TYPE
    ST_PickPlaceDetail : STRUCT
        MemberType : STRING;
        XPos       : REAL;
        YPos       : REAL;
        ZPos       : REAL;
        ZRot       : REAL;
        ConvIndex  : INT;
    END_STRUCT
END_TYPE

(* stored: Version 1.1.0.1
   DUT ST_PickPlaceDetail: Id {2a428ba2-0976-45e1-bb0d-92f7b4b6cd0f} *)
